FUNCTION_BLOCK Unifilar (* Composite Function Block Type *)
  (* Standard: 61499-2 *)
  (* Version 0.0, 21/04/2026, template *)
  PACKAGE Hidryco.HidrycoLib;
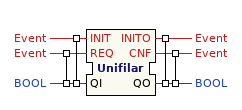
  EVENT_INPUT
    INIT WITH QI; (* Initialization Request *)
    REQ WITH QI; (* Normal Execution Request *)
  END_EVENT
  EVENT_OUTPUT
    INITO WITH QO; (* Initialization Confirm *)
    CNF WITH QO; (* Execution Confirmation *)
  END_EVENT
  VAR_INPUT
    QI : BOOL; (* Input event qualifier *)
  END_VAR
  VAR_OUTPUT
    QO : BOOL; (* Output event qualifier *)
  END_VAR
  FBS
    SYMLINKMULTIVARDST1 : SYMLINKMULTIVARDST_854A896E88500D19(NAME1 := '$${PATH}PCE_DisjuntorLigado', NAME2 := '$${PATH}V4603_DisjuntorLigado', NAME3 := '$${PATH}V4604_DisjuntorLigado', NAME4 := '$${PATH}COMP_500_02_DisjuntorLigado', NAME5 := '$${PATH}UCT_200_01_DisjuntorLigado', NAME6 := '$${PATH}PCM_EEE_BRUTO_DisjuntorLigado', NAME7 := '$${PATH}QGBT_220V_DisjuntorLigado', NAME8 := '$${PATH}PCM_DESINFECCAO_DisjuntorLigado', NAME9 := '$${PATH}BANCO_CAPACITORES_DisjuntorLigado', NAME10 := '$${PATH}V4601_DisjuntorLigado', NAME11 := '$${PATH}V4602_DisjuntorLigado', NAME12 := '$${PATH}COMP_500_01_DisjuntorLigado', NAME13 := '$${PATH}UCT_200_02_DisjuntorLigado', NAME14 := '$${PATH}UCT_200_03_DisjuntorLigado', NAME15 := '$${PATH}PCM_NER_DisjuntorLigado', NAME16 := '$${PATH}PCM_LD_DisjuntorLigado'); {SET_ATTRIBUTE(Configuration.GenericFBType.InterfaceParams, Runtime.System#I:=16;VALUE${I$}:BOOL,BOOL,BOOL,BOOL,BOOL,BOOL,BOOL,BOOL,BOOL,BOOL,BOOL,BOOL,BOOL,BOOL,BOOL,BOOL)}
    SYMLINKMULTIVARDST2 : SYMLINKMULTIVARDST_854A896E88500D19(NAME1 := '$${PATH}CAP2_DisjuntorLigado', NAME2 := '$${PATH}QBGT_220V_DisjuntorLigado', NAME3 := '$${PATH}QL_ADM_DisjuntorLigado', NAME4 := '$${PATH}QL_PORTARIA_DisjuntorLigado', NAME5 := '$${PATH}QLSL_DisjuntorLigado', NAME6 := '$${PATH}QL_ILUMINACAO_DisjuntorLigado', NAME7 := '$${PATH}PCE_SOPRADORES_DisjuntorLigado', NAME8 := '$${PATH}QL_LODO_DisjuntorLigado', NAME9 := '$${PATH}PCM_AGUA_REUSO_DisjuntorLigado', NAME10 := '$${PATH}CO_100_01_DisjuntorLigado', NAME11 := '$${PATH}CO_100_02_DisjuntorLigado', NAME12 := '$${PATH}CO_100_03_DisjuntorLigado', NAME13 := '$${PATH}CO_100_04_DisjuntorLigado', NAME14 := '$${PATH}GM_100_01_02_DisjuntorLigado', NAME15 := '$${PATH}MO_100_01_DisjuntorLigado', NAME16 := '$${PATH}UV_700_01_DisjuntorLigado'); {SET_ATTRIBUTE(Configuration.GenericFBType.InterfaceParams, Runtime.System#I:=16;VALUE${I$}:BOOL,BOOL,BOOL,BOOL,BOOL,BOOL,BOOL,BOOL,BOOL,BOOL,BOOL,BOOL,BOOL,BOOL,BOOL,BOOL)}
    SYMLINKMULTIVARDST3 : SYMLINKMULTIVARDST_854A896E88500D19(NAME1 := '$${PATH}UV_700_02_DisjuntorLigado', NAME2 := '$${PATH}VC_700_01_DisjuntorLigado', NAME3 := '$${PATH}MO_700_01_DisjuntorLigado', NAME4 := '$${PATH}MO_300_01_DisjuntorLigado', NAME5 := '$${PATH}R4005A_DisjuntorLigado', NAME6 := '$${PATH}R4005B_DisjuntorLigado', NAME7 := '$${PATH}P4901_DisjuntorLigado', NAME8 := '$${PATH}P4902_DisjuntorLigado', NAME9 := '$${PATH}P4903_DisjuntorLigado', NAME10 := '$${PATH}SO_900_01_DisjuntorLigado', NAME11 := '$${PATH}SO_900_02_DisjuntorLigado', NAME12 := '$${PATH}AD_900_01_DisjuntorLigado', NAME13 := '$${PATH}AD_900_02_DisjuntorLigado', NAME14 := '$${PATH}AD_900_03_DisjuntorLigado', NAME15 := '$${PATH}PP_900_01_DisjuntorLigado', NAME16 := '$${PATH}MN_900_01_DisjuntorLigado'); {SET_ATTRIBUTE(Configuration.GenericFBType.InterfaceParams, Runtime.System#I:=16;VALUE${I$}:BOOL,BOOL,BOOL,BOOL,BOOL,BOOL,BOOL,BOOL,BOOL,BOOL,BOOL,BOOL,BOOL,BOOL,BOOL,BOOL)}
    SYMLINKMULTIVARDST4 : SYMLINKMULTIVARDST_854A896E88500D19(NAME1 := '$${PATH}MN_900_02_DisjuntorLigado', NAME2 := '$${PATH}MN_900_03_DisjuntorLigado', NAME3 := '$${PATH}MN_900_04_DisjuntorLigado', NAME4 := '$${PATH}MN_900_05_DisjuntorLigado', NAME5 := '$${PATH}BO_900_01_DisjuntorLigado', NAME6 := '$${PATH}BO_900_02_DisjuntorLigado', NAME7 := '$${PATH}BO_900_03_DisjuntorLigado', NAME8 := '$${PATH}BR_900_01_DisjuntorLigado', NAME9 := '$${PATH}BR_900_02_DisjuntorLigado', NAME10 := '$${PATH}VA_900_01_DisjuntorLigado', NAME11 := '$${PATH}VA_900_02_DisjuntorLigado', NAME12 := '$${PATH}VE_900_01_DisjuntorLigado', NAME13 := '$${PATH}VA_900_06_DisjuntorLigado', NAME14 := '$${PATH}VA_900_07_DisjuntorLigado', NAME15 := '$${PATH}VA_900_08_DisjuntorLigado', NAME16 := '$${PATH}VA_900_09_DisjuntorLigado'); {SET_ATTRIBUTE(Configuration.GenericFBType.InterfaceParams, Runtime.System#I:=16;VALUE${I$}:BOOL,BOOL,BOOL,BOOL,BOOL,BOOL,BOOL,BOOL,BOOL,BOOL,BOOL,BOOL,BOOL,BOOL,BOOL,BOOL)}
    SYMLINKMULTIVARDST5 : SYMLINKMULTIVARDST_854A896E88500D19(NAME1 := '$${PATH}VA_900_10_DisjuntorLigado', NAME2 := '$${PATH}VA_900_11_DisjuntorLigado', NAME3 := '$${PATH}VA_900_12_DisjuntorLigado', NAME4 := '$${PATH}VA_900_13_DisjuntorLigado', NAME5 := '$${PATH}VB_900_03_DisjuntorLigado', NAME6 := '$${PATH}VB_900_04_DisjuntorLigado', NAME7 := '$${PATH}MO_500_01', NAME8 := '$${PATH}PCM_AR', NAME9 := '$${PATH}VE_900_02', NAME10 := '$${PATH}PCE_EEE_BRUTO', NAME11 := '$${PATH}PCE_LODO', NAME12 := '$${PATH}PCE_NEREDA', NAME13 := '$${PATH}PCE_DESINFECCAO', NAME14 := '$${PATH}PCE_SUBSTACAO'); {SET_ATTRIBUTE(Configuration.GenericFBType.InterfaceParams, Runtime.System#I:=16;VALUE${I$}:BOOL,BOOL,BOOL,BOOL,BOOL,BOOL,BOOL,BOOL,BOOL,BOOL,BOOL,BOOL,BOOL,BOOL,BOOL,BOOL)}
    PCE : DisjuntorCAT;
    V4603 : DisjuntorCAT;
    V4604 : DisjuntorCAT;
    COMP_500_02 : DisjuntorCAT;
    UCT_200_01 : DisjuntorCAT;
    PCM_EEE_BRUTO : DisjuntorCAT;
    QGBT_220V : DisjuntorCAT;
    PCM_DESINFECCAO : DisjuntorCAT;
    BANCO_CAPACITORES : DisjuntorCAT;
    V4601 : DisjuntorCAT;
    V4602 : DisjuntorCAT;
    COMP_500_01 : DisjuntorCAT;
    UCT_200_02 : DisjuntorCAT;
    UCT_200_03 : DisjuntorCAT;
    PCM_NER : DisjuntorCAT;
    PCM_LD : DisjuntorCAT;
    CAP2 : DisjuntorCAT;
    QBGT_220V : DisjuntorCAT;
    QL_ADM : DisjuntorCAT;
    QL_PORTARIA : DisjuntorCAT;
    QLSL : DisjuntorCAT;
    QL_ILUMINACAO : DisjuntorCAT;
    PCE_SOPRADORES : DisjuntorCAT;
    QL_LODO : DisjuntorCAT;
    PCM_AGUA_REUSO : DisjuntorCAT;
    CO_100_01 : DisjuntorCAT;
    CO_100_02 : DisjuntorCAT;
    CO_100_03 : DisjuntorCAT;
    CO_100_04 : DisjuntorCAT;
    GM_100_01_02 : DisjuntorCAT;
    MO_100_01 : DisjuntorCAT;
    UV_700_01 : DisjuntorCAT;
    UV_700_02 : DisjuntorCAT;
    VC_700_01 : DisjuntorCAT;
    MO_700_01 : DisjuntorCAT;
    MO_300_01 : DisjuntorCAT;
    R4005A : DisjuntorCAT;
    R4005B : DisjuntorCAT;
    P4901 : DisjuntorCAT;
    P4902 : DisjuntorCAT;
    P4903 : DisjuntorCAT;
    SO_900_01 : DisjuntorCAT;
    SO_900_02 : DisjuntorCAT;
    AD_900_01 : DisjuntorCAT;
    AD_900_02 : DisjuntorCAT;
    AD_900_03 : DisjuntorCAT;
    PP_900_01 : DisjuntorCAT;
    MN_900_01 : DisjuntorCAT;
    MN_900_02 : DisjuntorCAT;
    MN_900_03 : DisjuntorCAT;
    MN_900_04 : DisjuntorCAT;
    MN_900_05 : DisjuntorCAT;
    BO_900_01 : DisjuntorCAT;
    BO_900_02 : DisjuntorCAT;
    BO_900_03 : DisjuntorCAT;
    BR_900_01 : DisjuntorCAT;
    BR_900_02 : DisjuntorCAT;
    VA_900_01 : DisjuntorCAT;
    VA_900_02 : DisjuntorCAT;
    VE_900_01 : DisjuntorCAT;
    VA_900_06 : DisjuntorCAT;
    VA_900_07 : DisjuntorCAT;
    VA_900_08 : DisjuntorCAT;
    VA_900_09 : DisjuntorCAT;
    VA_900_10 : DisjuntorCAT;
    VA_900_11 : DisjuntorCAT;
    VA_900_12 : DisjuntorCAT;
    VA_900_13 : DisjuntorCAT;
    VB_900_03 : DisjuntorCAT;
    VB_900_04 : DisjuntorCAT;
    MO_500_01 : DisjuntorCAT;
    PCM_AR : DisjuntorCAT;
    VE_900_02 : DisjuntorCAT;
    PCE_EEE_BRUTO : DisjuntorCAT;
    PCE_LODO : DisjuntorCAT;
    PCE_DESINFECCAO : DisjuntorCAT;
    PCE_NEREDA : DisjuntorCAT;
    PCE_SUBSTACAO : DisjuntorCAT;
    IThis : Unifilar_HMI;
  END_FBS
  EVENT_CONNECTIONS
    PCE.INITO TO V4603.INIT;
    V4603.INITO TO V4604.INIT;
    V4604.INITO TO COMP_500_02.INIT;
    COMP_500_02.INITO TO UCT_200_01.INIT;
    UCT_200_01.INITO TO PCM_EEE_BRUTO.INIT;
    PCM_EEE_BRUTO.INITO TO QGBT_220V.INIT;
    QGBT_220V.INITO TO PCM_DESINFECCAO.INIT;
    PCM_DESINFECCAO.INITO TO BANCO_CAPACITORES.INIT;
    BANCO_CAPACITORES.INITO TO V4601.INIT;
    V4601.INITO TO V4602.INIT;
    V4602.INITO TO COMP_500_01.INIT;
    COMP_500_01.INITO TO UCT_200_02.INIT;
    UCT_200_02.INITO TO UCT_200_03.INIT;
    UCT_200_03.INITO TO PCM_NER.INIT;
    PCM_NER.INITO TO PCM_LD.INIT;
    PCM_LD.INITO TO CAP2.INIT;
    CAP2.INITO TO QBGT_220V.INIT;
    QBGT_220V.INITO TO QL_ADM.INIT;
    QL_ADM.INITO TO QL_PORTARIA.INIT;
    QL_PORTARIA.INITO TO QLSL.INIT;
    QLSL.INITO TO QL_ILUMINACAO.INIT;
    QL_ILUMINACAO.INITO TO PCE_SOPRADORES.INIT;
    PCE_SOPRADORES.INITO TO QL_LODO.INIT;
    QL_LODO.INITO TO PCM_AGUA_REUSO.INIT;
    PCM_AGUA_REUSO.INITO TO CO_100_01.INIT;
    CO_100_01.INITO TO CO_100_02.INIT;
    CO_100_02.INITO TO CO_100_03.INIT;
    CO_100_03.INITO TO CO_100_04.INIT;
    CO_100_04.INITO TO GM_100_01_02.INIT;
    GM_100_01_02.INITO TO MO_100_01.INIT;
    MO_100_01.INITO TO UV_700_01.INIT;
    UV_700_01.INITO TO UV_700_02.INIT;
    UV_700_02.INITO TO VC_700_01.INIT;
    VC_700_01.INITO TO MO_700_01.INIT;
    MO_700_01.INITO TO MO_300_01.INIT;
    MO_300_01.INITO TO R4005A.INIT;
    R4005A.INITO TO R4005B.INIT;
    R4005B.INITO TO P4901.INIT;
    P4901.INITO TO P4902.INIT;
    P4902.INITO TO P4903.INIT;
    P4903.INITO TO SO_900_01.INIT;
    SO_900_01.INITO TO SO_900_02.INIT;
    SO_900_02.INITO TO AD_900_01.INIT;
    AD_900_01.INITO TO AD_900_02.INIT;
    AD_900_02.INITO TO AD_900_03.INIT;
    AD_900_03.INITO TO PP_900_01.INIT;
    PP_900_01.INITO TO MN_900_01.INIT;
    MN_900_01.INITO TO MN_900_02.INIT;
    MN_900_02.INITO TO MN_900_03.INIT;
    MN_900_03.INITO TO MN_900_04.INIT;
    MN_900_04.INITO TO MN_900_05.INIT;
    MN_900_05.INITO TO BO_900_01.INIT;
    BO_900_01.INITO TO BO_900_02.INIT;
    BO_900_02.INITO TO BO_900_03.INIT;
    BO_900_03.INITO TO BR_900_01.INIT;
    BR_900_01.INITO TO BR_900_02.INIT;
    BR_900_02.INITO TO VA_900_01.INIT;
    VA_900_01.INITO TO VA_900_02.INIT;
    VA_900_02.INITO TO VE_900_01.INIT;
    VE_900_01.INITO TO VA_900_06.INIT;
    VA_900_06.INITO TO VA_900_07.INIT;
    VA_900_07.INITO TO VA_900_08.INIT;
    VA_900_08.INITO TO VA_900_09.INIT;
    VA_900_09.INITO TO VA_900_10.INIT;
    VA_900_10.INITO TO VA_900_11.INIT;
    VA_900_11.INITO TO VA_900_12.INIT;
    VA_900_12.INITO TO VA_900_13.INIT;
    VA_900_13.INITO TO VB_900_03.INIT;
    VB_900_03.INITO TO VB_900_04.INIT;
    PCE_SUBSTACAO.INITO TO INITO;
    PCE.CNF TO V4603.REQ;
    V4603.CNF TO V4604.REQ;
    V4604.CNF TO COMP_500_02.REQ;
    COMP_500_02.CNF TO UCT_200_01.REQ;
    UCT_200_01.CNF TO PCM_EEE_BRUTO.REQ;
    PCM_EEE_BRUTO.CNF TO QGBT_220V.REQ;
    QGBT_220V.CNF TO PCM_DESINFECCAO.REQ;
    PCM_DESINFECCAO.CNF TO BANCO_CAPACITORES.REQ;
    BANCO_CAPACITORES.CNF TO V4601.REQ;
    V4601.CNF TO V4602.REQ;
    V4602.CNF TO COMP_500_01.REQ;
    COMP_500_01.CNF TO UCT_200_02.REQ;
    UCT_200_02.CNF TO UCT_200_03.REQ;
    UCT_200_03.CNF TO PCM_NER.REQ;
    PCM_NER.CNF TO PCM_LD.REQ;
    PCM_LD.CNF TO CAP2.REQ;
    CAP2.CNF TO QBGT_220V.REQ;
    QBGT_220V.CNF TO QL_ADM.REQ;
    QL_ADM.CNF TO QL_PORTARIA.REQ;
    QL_PORTARIA.CNF TO QLSL.REQ;
    QLSL.CNF TO QL_ILUMINACAO.REQ;
    QL_ILUMINACAO.CNF TO PCE_SOPRADORES.REQ;
    PCE_SOPRADORES.CNF TO QL_LODO.REQ;
    QL_LODO.CNF TO PCM_AGUA_REUSO.REQ;
    PCM_AGUA_REUSO.CNF TO CO_100_01.REQ;
    CO_100_01.CNF TO CO_100_02.REQ;
    CO_100_02.CNF TO CO_100_03.REQ;
    CO_100_03.CNF TO CO_100_04.REQ;
    CO_100_04.CNF TO GM_100_01_02.REQ;
    GM_100_01_02.CNF TO MO_100_01.REQ;
    MO_100_01.CNF TO UV_700_01.REQ;
    UV_700_01.CNF TO UV_700_02.REQ;
    UV_700_02.CNF TO VC_700_01.REQ;
    VC_700_01.CNF TO MO_700_01.REQ;
    MO_700_01.CNF TO MO_300_01.REQ;
    MO_300_01.CNF TO R4005A.REQ;
    R4005A.CNF TO R4005B.REQ;
    R4005B.CNF TO P4901.REQ;
    P4901.CNF TO P4902.REQ;
    P4902.CNF TO P4903.REQ;
    P4903.CNF TO SO_900_01.REQ;
    SO_900_01.CNF TO SO_900_02.REQ;
    SO_900_02.CNF TO AD_900_01.REQ;
    AD_900_01.CNF TO AD_900_02.REQ;
    AD_900_02.CNF TO AD_900_03.REQ;
    AD_900_03.CNF TO PP_900_01.REQ;
    PP_900_01.CNF TO MN_900_01.REQ;
    MN_900_01.CNF TO MN_900_02.REQ;
    MN_900_02.CNF TO MN_900_03.REQ;
    MN_900_03.CNF TO MN_900_04.REQ;
    MN_900_04.CNF TO MN_900_05.REQ;
    MN_900_05.CNF TO BO_900_01.REQ;
    BO_900_01.CNF TO BO_900_02.REQ;
    BO_900_02.CNF TO BO_900_03.REQ;
    BO_900_03.CNF TO BR_900_01.REQ;
    BR_900_01.CNF TO BR_900_02.REQ;
    BR_900_02.CNF TO VA_900_01.REQ;
    VA_900_01.CNF TO VA_900_02.REQ;
    VA_900_02.CNF TO VE_900_01.REQ;
    VE_900_01.CNF TO VA_900_06.REQ;
    VA_900_06.CNF TO VA_900_07.REQ;
    VA_900_07.CNF TO VA_900_08.REQ;
    VA_900_08.CNF TO VA_900_09.REQ;
    VA_900_09.CNF TO VA_900_10.REQ;
    VA_900_10.CNF TO VA_900_11.REQ;
    VA_900_11.CNF TO VA_900_12.REQ;
    VA_900_12.CNF TO VA_900_13.REQ;
    VA_900_13.CNF TO VB_900_03.REQ;
    VB_900_03.CNF TO VB_900_04.REQ;
    PCE_SUBSTACAO.CNF TO CNF;
    INIT TO SYMLINKMULTIVARDST1.INIT;
    REQ TO SYMLINKMULTIVARDST1.REQ;
    SYMLINKMULTIVARDST1.INITO TO SYMLINKMULTIVARDST2.INIT;
    SYMLINKMULTIVARDST1.CNF TO SYMLINKMULTIVARDST2.REQ;
    SYMLINKMULTIVARDST2.INITO TO SYMLINKMULTIVARDST3.INIT;
    SYMLINKMULTIVARDST2.CNF TO SYMLINKMULTIVARDST3.REQ;
    SYMLINKMULTIVARDST3.INITO TO SYMLINKMULTIVARDST4.INIT;
    SYMLINKMULTIVARDST3.CNF TO SYMLINKMULTIVARDST4.REQ;
    VB_900_04.INITO TO MO_500_01.INIT;
    VB_900_04.CNF TO MO_500_01.REQ;
    MO_500_01.INITO TO VE_900_02.INIT;
    MO_500_01.CNF TO VE_900_02.REQ;
    SYMLINKMULTIVARDST4.INITO TO SYMLINKMULTIVARDST5.INIT;
    SYMLINKMULTIVARDST4.CNF TO SYMLINKMULTIVARDST5.REQ;
    SYMLINKMULTIVARDST5.INITO TO PCE.INIT;
    SYMLINKMULTIVARDST5.CNF TO PCE.REQ;
    VE_900_02.INITO TO PCE_EEE_BRUTO.INIT;
    VE_900_02.CNF TO PCE_EEE_BRUTO.REQ;
    PCE_EEE_BRUTO.INITO TO PCE_LODO.INIT;
    PCE_EEE_BRUTO.CNF TO PCE_LODO.REQ;
    PCE_LODO.INITO TO PCE_DESINFECCAO.INIT;
    PCE_LODO.CNF TO PCE_DESINFECCAO.REQ;
    PCE_DESINFECCAO.INITO TO PCE_NEREDA.INIT;
    PCE_DESINFECCAO.CNF TO PCE_NEREDA.REQ;
    PCE_NEREDA.INITO TO PCE_SUBSTACAO.INIT;
    PCE_NEREDA.CNF TO PCE_SUBSTACAO.REQ;
  END_CONNECTIONS
  DATA_CONNECTIONS
    QI TO PCE.QI;
    QI TO V4603.QI;
    QI TO V4604.QI;
    QI TO COMP_500_02.QI;
    QI TO UCT_200_01.QI;
    QI TO PCM_EEE_BRUTO.QI;
    QI TO QGBT_220V.QI;
    QI TO PCM_DESINFECCAO.QI;
    QI TO BANCO_CAPACITORES.QI;
    QI TO V4601.QI;
    QI TO V4602.QI;
    QI TO COMP_500_01.QI;
    QI TO UCT_200_02.QI;
    QI TO UCT_200_03.QI;
    QI TO PCM_NER.QI;
    QI TO PCM_LD.QI;
    QI TO CAP2.QI;
    QI TO QBGT_220V.QI;
    QI TO QL_ADM.QI;
    QI TO QL_PORTARIA.QI;
    QI TO QLSL.QI;
    QI TO QL_ILUMINACAO.QI;
    QI TO PCE_SOPRADORES.QI;
    QI TO QL_LODO.QI;
    QI TO PCM_AGUA_REUSO.QI;
    QI TO CO_100_01.QI;
    QI TO CO_100_02.QI;
    QI TO CO_100_03.QI;
    QI TO CO_100_04.QI;
    QI TO GM_100_01_02.QI;
    QI TO MO_100_01.QI;
    QI TO UV_700_01.QI;
    QI TO UV_700_02.QI;
    QI TO VC_700_01.QI;
    QI TO MO_700_01.QI;
    QI TO MO_300_01.QI;
    QI TO R4005A.QI;
    QI TO R4005B.QI;
    QI TO P4901.QI;
    QI TO P4902.QI;
    QI TO P4903.QI;
    QI TO SO_900_01.QI;
    QI TO SO_900_02.QI;
    QI TO AD_900_01.QI;
    QI TO AD_900_02.QI;
    QI TO AD_900_03.QI;
    QI TO PP_900_01.QI;
    QI TO MN_900_01.QI;
    QI TO MN_900_02.QI;
    QI TO MN_900_03.QI;
    QI TO MN_900_04.QI;
    QI TO MN_900_05.QI;
    QI TO BO_900_01.QI;
    QI TO BO_900_02.QI;
    QI TO BO_900_03.QI;
    QI TO BR_900_01.QI;
    QI TO BR_900_02.QI;
    QI TO VA_900_01.QI;
    QI TO VA_900_02.QI;
    QI TO VE_900_01.QI;
    QI TO VA_900_06.QI;
    QI TO VA_900_07.QI;
    QI TO VA_900_08.QI;
    QI TO VA_900_09.QI;
    QI TO VA_900_10.QI;
    QI TO VA_900_11.QI;
    QI TO VA_900_12.QI;
    QI TO VA_900_13.QI;
    QI TO VB_900_03.QI;
    QI TO VB_900_04.QI;
    QI TO SYMLINKMULTIVARDST1.QI;
    SYMLINKMULTIVARDST1.VALUE1 TO PCE.stsDisjuntorLigado;
    SYMLINKMULTIVARDST1.VALUE2 TO V4603.stsDisjuntorLigado;
    SYMLINKMULTIVARDST1.VALUE3 TO V4604.stsDisjuntorLigado;
    SYMLINKMULTIVARDST1.VALUE4 TO COMP_500_02.stsDisjuntorLigado;
    SYMLINKMULTIVARDST1.VALUE5 TO UCT_200_01.stsDisjuntorLigado;
    SYMLINKMULTIVARDST1.VALUE6 TO PCM_EEE_BRUTO.stsDisjuntorLigado;
    SYMLINKMULTIVARDST1.VALUE7 TO QGBT_220V.stsDisjuntorLigado;
    SYMLINKMULTIVARDST1.VALUE8 TO PCM_DESINFECCAO.stsDisjuntorLigado;
    SYMLINKMULTIVARDST1.VALUE9 TO BANCO_CAPACITORES.stsDisjuntorLigado;
    SYMLINKMULTIVARDST1.VALUE10 TO V4601.stsDisjuntorLigado;
    SYMLINKMULTIVARDST1.VALUE11 TO V4602.stsDisjuntorLigado;
    SYMLINKMULTIVARDST1.VALUE12 TO COMP_500_01.stsDisjuntorLigado;
    SYMLINKMULTIVARDST1.VALUE13 TO UCT_200_02.stsDisjuntorLigado;
    SYMLINKMULTIVARDST1.VALUE14 TO UCT_200_03.stsDisjuntorLigado;
    SYMLINKMULTIVARDST1.VALUE15 TO PCM_NER.stsDisjuntorLigado;
    SYMLINKMULTIVARDST1.VALUE16 TO PCM_LD.stsDisjuntorLigado;
    QI TO SYMLINKMULTIVARDST2.QI;
    SYMLINKMULTIVARDST2.VALUE1 TO CAP2.stsDisjuntorLigado;
    SYMLINKMULTIVARDST2.VALUE2 TO QBGT_220V.stsDisjuntorLigado;
    SYMLINKMULTIVARDST2.VALUE3 TO QL_ADM.stsDisjuntorLigado;
    SYMLINKMULTIVARDST2.VALUE4 TO QL_PORTARIA.stsDisjuntorLigado;
    SYMLINKMULTIVARDST2.VALUE5 TO QLSL.stsDisjuntorLigado;
    SYMLINKMULTIVARDST2.VALUE6 TO QL_ILUMINACAO.stsDisjuntorLigado;
    SYMLINKMULTIVARDST2.VALUE7 TO PCE_SOPRADORES.stsDisjuntorLigado;
    SYMLINKMULTIVARDST2.VALUE8 TO QL_LODO.stsDisjuntorLigado;
    SYMLINKMULTIVARDST2.VALUE9 TO PCM_AGUA_REUSO.stsDisjuntorLigado;
    SYMLINKMULTIVARDST2.VALUE10 TO CO_100_01.stsDisjuntorLigado;
    SYMLINKMULTIVARDST2.VALUE11 TO CO_100_02.stsDisjuntorLigado;
    SYMLINKMULTIVARDST2.VALUE12 TO CO_100_03.stsDisjuntorLigado;
    SYMLINKMULTIVARDST2.VALUE13 TO CO_100_04.stsDisjuntorLigado;
    SYMLINKMULTIVARDST2.VALUE14 TO GM_100_01_02.stsDisjuntorLigado;
    SYMLINKMULTIVARDST2.VALUE15 TO MO_100_01.stsDisjuntorLigado;
    SYMLINKMULTIVARDST2.VALUE16 TO UV_700_01.stsDisjuntorLigado;
    QI TO SYMLINKMULTIVARDST3.QI;
    SYMLINKMULTIVARDST3.VALUE1 TO UV_700_02.stsDisjuntorLigado;
    SYMLINKMULTIVARDST3.VALUE2 TO VC_700_01.stsDisjuntorLigado;
    SYMLINKMULTIVARDST3.VALUE3 TO MO_700_01.stsDisjuntorLigado;
    SYMLINKMULTIVARDST3.VALUE4 TO MO_300_01.stsDisjuntorLigado;
    SYMLINKMULTIVARDST3.VALUE5 TO R4005A.stsDisjuntorLigado;
    SYMLINKMULTIVARDST3.VALUE6 TO R4005B.stsDisjuntorLigado;
    SYMLINKMULTIVARDST3.VALUE7 TO P4901.stsDisjuntorLigado;
    SYMLINKMULTIVARDST3.VALUE8 TO P4902.stsDisjuntorLigado;
    SYMLINKMULTIVARDST3.VALUE9 TO P4903.stsDisjuntorLigado;
    SYMLINKMULTIVARDST3.VALUE10 TO SO_900_01.stsDisjuntorLigado;
    SYMLINKMULTIVARDST3.VALUE11 TO SO_900_02.stsDisjuntorLigado;
    SYMLINKMULTIVARDST3.VALUE12 TO AD_900_01.stsDisjuntorLigado;
    SYMLINKMULTIVARDST3.VALUE13 TO AD_900_02.stsDisjuntorLigado;
    SYMLINKMULTIVARDST3.VALUE14 TO AD_900_03.stsDisjuntorLigado;
    SYMLINKMULTIVARDST3.VALUE15 TO PP_900_01.stsDisjuntorLigado;
    SYMLINKMULTIVARDST3.VALUE16 TO MN_900_01.stsDisjuntorLigado;
    QI TO SYMLINKMULTIVARDST4.QI;
    SYMLINKMULTIVARDST4.VALUE1 TO MN_900_02.stsDisjuntorLigado;
    SYMLINKMULTIVARDST4.VALUE2 TO MN_900_03.stsDisjuntorLigado;
    SYMLINKMULTIVARDST4.VALUE3 TO MN_900_04.stsDisjuntorLigado;
    SYMLINKMULTIVARDST4.VALUE4 TO MN_900_05.stsDisjuntorLigado;
    SYMLINKMULTIVARDST4.VALUE5 TO BO_900_01.stsDisjuntorLigado;
    SYMLINKMULTIVARDST4.VALUE6 TO BO_900_02.stsDisjuntorLigado;
    SYMLINKMULTIVARDST4.VALUE7 TO BO_900_03.stsDisjuntorLigado;
    SYMLINKMULTIVARDST4.VALUE8 TO BR_900_01.stsDisjuntorLigado;
    SYMLINKMULTIVARDST4.VALUE9 TO BR_900_02.stsDisjuntorLigado;
    SYMLINKMULTIVARDST4.VALUE10 TO VA_900_01.stsDisjuntorLigado;
    SYMLINKMULTIVARDST4.VALUE11 TO VA_900_02.stsDisjuntorLigado;
    SYMLINKMULTIVARDST4.VALUE12 TO VE_900_01.stsDisjuntorLigado;
    SYMLINKMULTIVARDST4.VALUE13 TO VA_900_06.stsDisjuntorLigado;
    SYMLINKMULTIVARDST4.VALUE14 TO VA_900_07.stsDisjuntorLigado;
    SYMLINKMULTIVARDST4.VALUE15 TO VA_900_08.stsDisjuntorLigado;
    SYMLINKMULTIVARDST4.VALUE16 TO VA_900_09.stsDisjuntorLigado;
    QI TO SYMLINKMULTIVARDST5.QI;
    SYMLINKMULTIVARDST5.VALUE1 TO VA_900_10.stsDisjuntorLigado;
    SYMLINKMULTIVARDST5.VALUE2 TO VA_900_11.stsDisjuntorLigado;
    SYMLINKMULTIVARDST5.VALUE3 TO VA_900_12.stsDisjuntorLigado;
    SYMLINKMULTIVARDST5.VALUE4 TO VA_900_13.stsDisjuntorLigado;
    SYMLINKMULTIVARDST5.VALUE5 TO VB_900_03.stsDisjuntorLigado;
    SYMLINKMULTIVARDST5.VALUE6 TO VB_900_04.stsDisjuntorLigado;
    SYMLINKMULTIVARDST5.VALUE7 TO MO_500_01.stsDisjuntorLigado;
    SYMLINKMULTIVARDST5.VALUE8 TO PCM_AR.stsDisjuntorLigado;
    SYMLINKMULTIVARDST5.VALUE9 TO VE_900_02.stsDisjuntorLigado;
    SYMLINKMULTIVARDST5.VALUE10 TO PCE_EEE_BRUTO.stsDisjuntorLigado;
    SYMLINKMULTIVARDST5.VALUE11 TO PCE_LODO.stsDisjuntorLigado;
    SYMLINKMULTIVARDST5.VALUE12 TO PCE_NEREDA.stsDisjuntorLigado;
    SYMLINKMULTIVARDST5.VALUE13 TO PCE_DESINFECCAO.stsDisjuntorLigado;
    SYMLINKMULTIVARDST5.VALUE14 TO PCE_SUBSTACAO.stsDisjuntorLigado;
    VA_900_01.QO TO IThis.FC63ECCCD56E3411;
    VA_900_02.QO TO IThis.F80C065CAA367883;
    VA_900_06.QO TO IThis.1B2A24A27E371AA3;
    VA_900_07.QO TO IThis.F6C968F0317F9E40;
    VA_900_10.QO TO IThis.899A54AD0C90C201;
    VA_900_11.QO TO IThis.FD6A2E53352C076C;
    VA_900_12.QO TO IThis.B631634C39D9FF5C;
    VA_900_13.QO TO IThis.93B3D5ED9A9F7176;
    VB_900_03.QO TO IThis.CE3E5851E0027041;
    VB_900_04.QO TO IThis.BEB680EBBFAABECA;
    VA_900_08.QO TO IThis.14819388827A4681;
    VA_900_09.QO TO IThis.1577BCBA9FF36EF5;
    BR_900_02.QO TO IThis.99517E0DFCA99F71;
    BR_900_01.QO TO IThis.10E062977E039F5D;
    BO_900_03.QO TO IThis.F2C782A461B41289;
    BO_900_02.QO TO IThis.11AD346572F7FDF;
    BO_900_01.QO TO IThis.A50730B8FE50C355;
    MN_900_05.QO TO IThis.6100EECBED531B79;
    MN_900_04.QO TO IThis.7F114654BE72541A;
    MN_900_03.QO TO IThis.B870E5D6CAA17BAD;
    MN_900_02.QO TO IThis.A22AC6AB9B6F2930;
    MN_900_01.QO TO IThis.30707D9D4AB84740;
    PP_900_01.QO TO IThis.D57B8A43F37D109E;
    AD_900_03.QO TO IThis.DE70CD4C348D950C;
    AD_900_02.QO TO IThis.9D4E14C6CD36CE98;
    AD_900_01.QO TO IThis.3338B11A9DC6A654;
    SO_900_02.QO TO IThis.5B275581F1385212;
    SO_900_01.QO TO IThis.AE4DFBBC97AEBD23;
    P4903.QO TO IThis.328D021CCE600CE7;
    P4902.QO TO IThis.350BA6E7F971F56C;
    P4901.QO TO IThis.105EC4C98FFC4D04;
    R4005B.QO TO IThis.F1FD4314C8565E77;
    R4005A.QO TO IThis.B4BDAF23A1F82D51;
    MO_300_01.QO TO IThis.9AD7175E705E4B8D;
    MO_700_01.QO TO IThis.DD2F95BA645ED624;
    VC_700_01.QO TO IThis.85D4B6B8EAD03818;
    UV_700_02.QO TO IThis.19F158622D1C12B0;
    UV_700_01.QO TO IThis.C86D99D9031BD02B;
    MO_100_01.QO TO IThis.7ED5DB7C4804A162;
    GM_100_01_02.QO TO IThis.CF03E1A96CFD2C9B;
    CO_100_04.QO TO IThis.34C2AB7B3670FDB1;
    CO_100_03.QO TO IThis.72BBEE12BAF63D73;
    CO_100_02.QO TO IThis.74AB8977488C226;
    CO_100_01.QO TO IThis.55821AFF40DE6312;
    PCM_AGUA_REUSO.QO TO IThis.DC313145E794A31D;
    QL_LODO.QO TO IThis.193F8FB90D88EED2;
    PCE_SOPRADORES.QO TO IThis.B304DE0F5D40D44C;
    QL_ILUMINACAO.QO TO IThis.B2B7956FB8813C6A;
    QLSL.QO TO IThis.C322FB6DD1D2B4E6;
    QL_PORTARIA.QO TO IThis.99336DCFB8F285E1;
    QL_ADM.QO TO IThis.D900B38B94401491;
    QBGT_220V.QO TO IThis.AB6361DDB926DE22;
    CAP2.QO TO IThis.E61C764290BEC977;
    PCM_LD.QO TO IThis.D3A5A9532AFEDB46;
    PCM_NER.QO TO IThis.A1BE6CA7C67352D6;
    UCT_200_03.QO TO IThis.497A608EA5530AC7;
    UCT_200_02.QO TO IThis.112254E5094DB119;
    COMP_500_01.QO TO IThis.E618ED00DACCED81;
    V4602.QO TO IThis.3F5EED4631AD29B7;
    V4601.QO TO IThis.25F6B39DFD88B319;
    BANCO_CAPACITORES.QO TO IThis.6410798DF6089F25;
    PCM_DESINFECCAO.QO TO IThis.92512E4B1B0DF01D;
    PCM_EEE_BRUTO.QO TO IThis.C96B753822C2CA0A;
    UCT_200_01.QO TO IThis.76DA179220260075;
    COMP_500_02.QO TO IThis.ECE8740725581E2B;
    V4604.QO TO IThis.FC9D85BBBCAEB9D4;
    V4603.QO TO IThis.5FB11A98F946C5FC;
  END_CONNECTIONS
END_FUNCTION_BLOCK
